TYPE TelemetryAccelerometersConfig :
STRUCT
	///Accelerometer box at the tube
	tube: TelemetryAccelerometerConfig;
END_STRUCT
END_TYPE

(* stored: Version 1.1.0.1, ProductVersion 3.1.4019.2
   DUT TelemetryAccelerometersConfig: Id {a743b112-e73e-40aa-bd7e-e858380f3557} *)
